// Mitsubishi GX Works2 project: 서보 모터 위치 티칭 (응용)   PLC: Q03UDV

PROGRAM MAIN
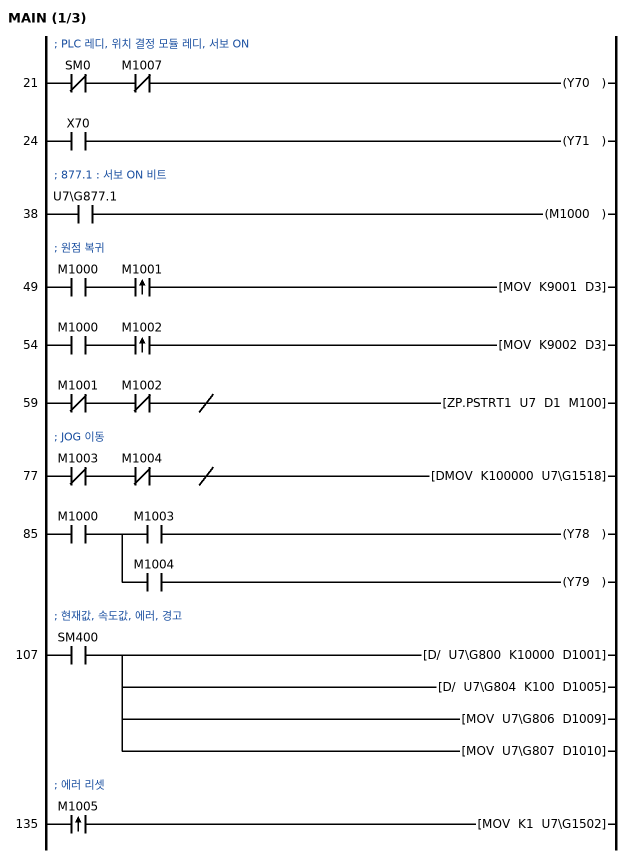
; PLC 레디, 위치 결정 모듈 레디, 서보 ON
21    LDI     SM0
      ANI     M1007
      OUT     Y70
24    LD      X70
      OUT     Y71
; 877.1 : 서보 ON 비트
38    LD      U7\G877.1
      OUT     M1000
; 원점 복귀
49    LD      M1000
      ANDP    M1001
      MOV     K9001 D3
54    LD      M1000
      ANDP    M1002
      MOV     K9002 D3
59    LDI     M1001
      ANI     M1002
      INV
      ZP.PSTRT1 U7 D1 M100
; JOG 이동
77    LDI     M1003
      ANI     M1004
      INV
      DMOV    K100000 U7\G1518
85    LD      M1000
      MPS
      AND     M1003
      OUT     Y78
      MPP
      AND     M1004
      OUT     Y79
; 현재값, 속도값, 에러, 경고
107   LD      SM400
      D/      U7\G800 K10000 D1001
      D/      U7\G804 K100 D1005
      MOV     U7\G806 D1009
      MOV     U7\G807 D1010
; 에러 리셋
135   LDP     M1005
      MOV     K1 U7\G1502
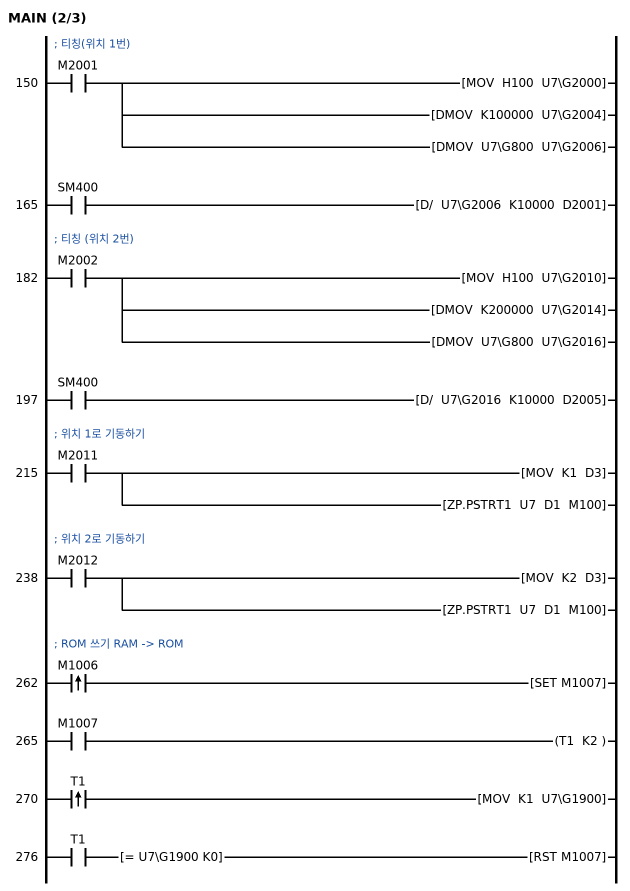
; 티칭(위치 1번)
150   LD      M2001
      MOV     H100 U7\G2000
      DMOV    K100000 U7\G2004
      DMOV    U7\G800 U7\G2006
165   LD      SM400
      D/      U7\G2006 K10000 D2001
; 티칭 (위치 2번)
182   LD      M2002
      MOV     H100 U7\G2010
      DMOV    K200000 U7\G2014
      DMOV    U7\G800 U7\G2016
197   LD      SM400
      D/      U7\G2016 K10000 D2005
; 위치 1로 기동하기
215   LD      M2011
      MOV     K1 D3
      ZP.PSTRT1 U7 D1 M100
; 위치 2로 기동하기
238   LD      M2012
      MOV     K2 D3
      ZP.PSTRT1 U7 D1 M100
; ROM 쓰기 RAM -> ROM
262   LDP     M1006
      SET     M1007
265   LD      M1007
      OUT     T1 K2
270   LDP     T1
      MOV     K1 U7\G1900
276   LD      T1
      AND=    U7\G1900 K0
      RST     M1007
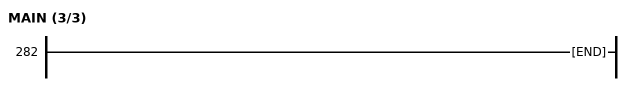
282   END
END_PROGRAM
